// TwinCAT 3 PLC project PLC
// ProgramVersion: 3.1.4023.0
// libraries:
//   Tc2_ControllerToolbox, * (Beckhoff Automation GmbH)
//   Tc2_EtherCAT, * (Beckhoff Automation GmbH)
//   Tc2_FTP, * (Beckhoff Automation GmbH)
//   Tc2_ModbusRTU, * (Beckhoff Automation GmbH)
//   Tc2_ModbusSrv, * (Beckhoff Automation GmbH)
//   Tc2_ProfinetDiag, * (Beckhoff Automation GmbH)
//   Tc2_Standard, * (Beckhoff Automation GmbH)
//   Tc2_SUPS, * (Beckhoff Automation GmbH)
//   Tc2_System, * (Beckhoff Automation GmbH)
//   Tc2_Utilities, * (Beckhoff Automation GmbH)
//   Tc3_EventLogger, * (Beckhoff Automation GmbH)
//   Tc3_IotBase, * (Beckhoff Automation GmbH)
//   Tc3_JsonXml, * (Beckhoff Automation GmbH)
//   Tc3_Module, * (Beckhoff Automation GmbH)
//   Base Interfaces,newest,System
// project tree:
//   DUTs/Enums/ eGridTripMode.TcDUT, eBatteryType.TcDUT, eObject_ID.TcDUT, ePNcouplerType.TcDUT, eSubValues.TcDUT, Phases.TcDUT
//   DUTs/Structs/ ST_AnalogInputData.TcDUT, ST_AnalogInputDiag.TcDUT
//   DUTs/System/ ST_System_Config.TcDUT, ST_System_GridcodeParams.TcDUT, ST_System_MachineParams.TcDUT
//   GVLs/ GVL.TcGVL, Settings.TcGVL, Units.TcGVL
//   / PlcTask.TcTTO, MonitorControlTask.TcTTO
//   POUs/Datalogger/DataLogging/ ArrayVariables.TcPOU, Datalogger.TcPOU, ST_Datalog_event.TcDUT
//   POUs/Datalogger/FUNCTIONBLOCKS/ FB_CSVWriter.TcPOU, FB_Datalogger.TcPOU, ToHexConverter.TcPOU
//   POUs/ErrorHandling/ ErrorHandling.TcPOU, FB_AddErrorST.TcPOU
//   POUs/ErrorHandling/New eventlogger %28TBD%29/ EventLogger.TcPOU (not stored), FB_Alarm.TcPOU (not stored), fb_EventAlarm.TcPOU (not stored)
//   POUs/ErrorHandling/_enums/ eErrAckAccess.TcDUT, eSeverity.TcDUT
//   POUs/ErrorHandling/_strucs/ ST_ErrorStruct.TcDUT
//   POUs/EventLogger/ EventLog.TcPOU (excluded from build), WriteLogItem.TcPOU (excluded from build)
//   POUs/EventLogger/_enums/ eLogSeverity.TcDUT
//   POUs/EventLogger/_Structs/ ST_EventLoggerParams.TcDUT
//   POUs/Functions-FBs-Programs/ Fb_BindControlVars.TcPOU, FB_OverCurrentDetect.TcPOU, fb_Ramp_dual.TcPOU, fbValueOutOfRange.TcPOU, fb_IncrementPowerStep.TcPOU, fb_Ramp.TcPOU, FB_UpperLimitAndTimeExceeded.TcPOU
//   POUs/Functions-FBs-Programs/IO_modules/Beckhoff/ FB_EK1100.TcPOU, FB_EL34xx.TcPOU, FB_EL3453.TcPOU
//   POUs/Functions-FBs-Programs/IO_modules/Beckhoff/Structs/ DataSelector.TcDUT, ST_EL34xx_PhaseStatus.TcDUT, ST_EL34xx_TotalStatus.TcDUT
//   POUs/Functions-FBs-Programs/IO_modules/Wago/ FB_Wago750354_BusCoupler.TcPOU, FB_Wago750495_PowerMonitor.TcPOU
//   POUs/Functions-FBs-Programs/IO_modules/Wago/Structs/Wago750354/ ST_Wago750354_get.TcDUT
//   POUs/Functions-FBs-Programs/IO_modules/Wago/Structs/Wago750495/ eWago750495_ACDataID.TcDUT, eWago750495_HarmonicsDataID.TcDUT, eWago750495_MeasureGroupID.TcDUT, eWago750495_StatDataID.TcDUT, ST_Wago750495_Data.TcDUT, ST_Wago750495_ExtStatusWord.TcDUT, ST_Wago750495_Get.TcDUT, ST_Wago750495_Set.TcDUT, ST_Wago750495_StatusWord.TcDUT
//   POUs/Functions-FBs-Programs/_acFunctions/ AcCheck.TcPOU, ACFrequencyCheck.TcPOU, ACVoltageCheck.TcPOU, CurrentToKw.TcPOU, fb_LOMdetection.TcPOU, kWToCurrent.TcPOU, LineUnbalance.TcPOU, PowerFactor.TcPOU, ReactivePower.TcPOU
//   POUs/Functions-FBs-Programs/_generalFunctions/ Between.TcPOU, ConcatMultiString.TcPOU, fb_MovingAverage.TcPOU, FB_StartStop.TcPOU, F_RoundReal.TcPOU, IsNaN.TcPOU, LimitTrigger.TcPOU, PackByte.TcPOU, PackWord.TcPOU, Median.TcPOU, Scale.TcPOU, ValueOutOfRange.TcPOU, WriteOnEdge.TcPOU, XNOR.TcPOU
//   POUs/Functions-FBs-Programs/_PRGS/ SystemClock.TcPOU
//   POUs/ MAIN_Fast.TcPOU, MAIN_Slow.TcPOU
//   POUs/MonitoringControl/ ControlManager.TcPOU, FB_TestScripts.TcPOU
//   POUs/MonitoringControl/HMI/ FB_HMIButtons.TcPOU, HMI.TcPOU
//   POUs/MonitoringControl/HMI/_Structs/ControlStructures/HardSettings %28localOnly%29/ ST_HardSettings.TcDUT (not stored), ST_HardSettings_DCcharger.TcDUT (not stored), ST_HardSettings_ParallelOperation.TcDUT (not stored), ST_HardSettings_PeakshaveBox.TcDUT (not stored), ST_HardSettings_Setup.TcDUT (not stored), ST_HardSettings_System.TcDUT (not stored)
//   POUs/MonitoringControl/HMI/_Structs/ControlStructures/OperationVars/ ST_OperationVars.TcDUT, ST_OperationVars_BMS.TcDUT, ST_OperationVars_DCcharger.TcDUT, ST_OperationVars_Genset.TcDUT, ST_OperationVars_Grid.TcDUT, ST_OperationVars_ParallelOperation.TcDUT, ST_OperationVars_System.TcDUT
//   POUs/MonitoringControl/HMI/_Structs/ControlStructures/SoftSettings %28Local+Extern%29/NestedStructs/ ST_Genset_params.TcDUT (not stored), ST_Genset_setpoints.TcDUT (not stored), ST_Input_breakersettings.TcDUT (not stored), ST_Loadbank_params.TcDUT (not stored), ST_peakshave_setpoints.TcDUT (not stored), ST_ScheduleTimeSlot.TcDUT (not stored)
//   POUs/MonitoringControl/HMI/_Structs/ControlStructures/SoftSettings %28Local+Extern%29/ ST_SoftSettings.TcDUT (not stored), ST_Softsettings_AcDcCharger.TcDUT (not stored), ST_SoftSettings_Genset.TcDUT (not stored), ST_SoftSettings_Grid.TcDUT (not stored), ST_SoftSettings_PeakshaveBox.TcDUT (not stored), ST_SoftSettings_Setup.TcDUT (not stored), ST_SoftSettings_System.TcDUT (not stored)
//   POUs/MonitoringControl/HMI/_Structs/ControlStructures/ ST_ControlsHMIonly.TcDUT, ST_ControlVars.TcDUT
//   POUs/MonitoringControl/HMI/_Structs/MonitoringStructures/ ST_HMIdata.TcDUT, ST_HMI_ConditionalFormatting.TcDUT, ST_HMI_Monitor_AcDcCharger.TcDUT, ST_HMI_Monitor_Arraydata.TcDUT, ST_HMI_Monitor_ArrayDataFormat.TcDUT, ST_HMI_Monitor_Connections.TcDUT, ST_HMI_Monitor_Battery.TcDUT, ST_HMI_Monitor_CoolingSystem.TcDUT, ST_HMI_Monitor_Enclosure.TcDUT, ST_HMI_Monitor_FireDetection.TcDUT, ST_HMI_Monitor_IPSU.TcDUT, ST_HMI_Monitor_Limits.TcDUT, ST_HMI_Monitor_OCP.TcDUT, ST_HMI_Monitor_Powerstack.TcDUT, ST_HMI_Monitor_Protections.TcDUT, ST_HMI_Monitor_PSB.TcDUT, ST_HMI_Monitor_switchgear.TcDUT, ST_HMI_Monitor_System.TcDUT, ST_HMI_Monitor_UPS.TcDUT, ST_HMI_Monitor_ZPT.TcDUT, ST_HMI_PowerMeas.TcDUT, ST_HMI_PowerMeasDC.TcDUT
//   POUs/MonitoringControl/HMI/_Structs/ ST_HMI_Control.TcDUT, ST_HMI_Historize.TcDUT, ST_HMI_Monitor.TcDUT
//   POUs/MonitoringControl/IoT/DUTS/ eConnectionState.TcDUT, eDataMappingVarNames.TcDUT, eIoTCommVersion.TcDUT, eLogType.TcDUT, eUpdate.TcDUT, e_ORAttributeType.TcDUT, ST_AutoProvisioning.TcDUT, ST_IotProps.TcDUT, ST_RW.TcDUT, ST_Supervisor.TcDUT, ST_VarBuffer.TcDUT
//   POUs/MonitoringControl/IoT/ FB_IotController.TcPOU, MqttComOpenremote.TcPOU, RestComOpenremote.TcPOU
//   POUs/MonitoringControl/IoT/_Structs/ ST_IoTDataHMI.TcDUT, ST_IotData_credits.TcDUT, st_IOT_params.TcDUT, ST_IOT_SentStateLog.TcDUT
//   POUs/MonitoringControl/ProfinetController/enums/ eExternalControlMode.TcDUT, GenGridMode.TcDUT, uSWversion.TcDUT
//   POUs/MonitoringControl/ProfinetController/ FB_ExtControllerTest.TcPOU, FB_ExternalController.TcPOU
//   POUs/MonitoringControl/ProfinetController/Structs/future use/ ST_PNInput_DCBusExpansion.TcDUT, ST_PNInput_DCCharger.TcDUT, ST_PNInput_ParallelOperation.TcDUT, ST_PNOutput_DCCharger.TcDUT, ST_PNOutput_DCExpansion.TcDUT, ST_PNOutput_ParallelOperation.TcDUT
//   POUs/MonitoringControl/ProfinetController/Structs/NestedStructs/ ST_PNInput_ACDCCharger.TcDUT, ST_PNInput_Battery.TcDUT, ST_PNInput_GenControl.TcDUT, ST_PNInput_General.TcDUT, ST_PNInput_InputField.TcDUT, ST_PNInput_InputGridControl.TcDUT, ST_PNInput_PeakShaveBox.TcDUT, ST_PNInput_Powerstack.TcDUT, ST_PNOutput_ACDCCharger.TcDUT, ST_PNOutput_Battery.TcDUT, ST_PNOutput_GenControl.TcDUT, ST_PNOutput_General.TcDUT, ST_PNOutput_InputField.TcDUT, ST_PNOutput_InputGridControl.TcDUT, ST_PNOutput_OutputField.TcDUT, ST_PNOutput_PeakShaveBox.TcDUT, ST_PNOutput_PowerStack.TcDUT, ST_PNOutput_ZPT.TcDUT
//   POUs/MonitoringControl/ProfinetController/Structs/ ST_PNcontroller_params.TcDUT, ST_PNinput.TcDUT, ST_PNOutput.TcDUT, ST_PNTest.TcDUT
//   POUs/MonitoringControl/_Enums/ eAcInputType.TcDUT, eCapTestSTate.TcDUT, eControlSources.TcDUT, eDcInputType.TcDUT, eEarthingSystems.TcDUT, eGridFormingMode.TcDUT, eGridMode.TcDUT, eNetContactorDirection.TcDUT, eOperationMode.TcDUT, ePeakshaveMode.TcDUT, eSchedulerMode.TcDUT, ePowerControlType.TcDUT, eSystemState.TcDUT, eUgridPowerMode.TcDUT
//   POUs/MonitoringControl/_Structs/ ST_ExtController_Events.TcDUT, ST_ExtController_get.TcDUT, ST_ExtController_limits.TcDUT, ST_ExtController_Set.TcDUT, ST_PLCPersistentVars.TcDUT
//   POUs/Objects/4Grouter/ FB_Teltonika.TcPOU
//   POUs/Objects/4Grouter/Struct/ dwtoreal.TcDUT, eModemState.TcDUT, eNetworkState.TcDUT, eSimSelectionMode.TcDUT, eSimState.TcDUT, eSMSStatus.TcDUT, eWifiSecurityTypes.TcDUT, eWifiStatus.TcDUT, st_Device.TcDUT, st_GPS.TcDUT, st_mobile.TcDUT, st_router_get.TcDUT, ST_Router_params.TcDUT, st_Router_Events.TcDUT, ST_Router_set.TcDUT, st_Wifi.TcDUT
//   POUs/Objects/ACDCCharger/Enums/ eAcDcChargerState.TcDUT
//   POUs/Objects/ACDCCharger/ FB_ACDCcharger.TcPOU
//   POUs/Objects/ACDCCharger/Structs/Hadi/ E_ChargerState.TcDUT, ST_CanId.TcDUT, ST_ChargerControl.TcDUT, ST_Control.TcDUT, ST_Data.TcDUT, ST_ModuleControl.TcDUT, ST_ModuleData.TcDUT, ST_ModuleStatus.TcDUT
//   POUs/Objects/ACDCCharger/Structs/ ST_ACDCCharger_events.TcDUT, ST_ACDCCharger_get.TcDUT, ST_ACDCCharger_params.TcDUT, ST_ACDCCharger_set.TcDUT, ST_SystemDiagnostic.TcDUT, ST_SystemEval.TcDUT
//   POUs/Objects/ACSwitchgear %28clientbox%29/ FB_ACSwitchgear.TcPOU (not stored), ST_ACswitchgear_events.TcDUT (not stored), ST_ACSwitchgear_Get.TcDUT (not stored), ST_ACswitchgear_IO.TcDUT (not stored), ST_ACswitchgear_params.TcDUT (not stored), ST_ACswitchgear_set.TcDUT (not stored)
//   POUs/Objects/BMS/eNums/ eBMS_Status.TcDUT, eHVDC_Powerstatus.TcDUT, ePOUState.TcDUT, ePowerControl.TcDUT, ePowerOnStatus.TcDUT
//   POUs/Objects/BMS/ FB_BMS.TcPOU, FB_BMS_IO.TcPOU
//   POUs/Objects/BMS/Structs/ st_BMS_Events.TcDUT, st_BMS_Get.TcDUT, st_BMS_Params.TcDUT, st_BMS_BatterySummary.TcDUT, st_BMS_Set.TcDUT, st_MBMU_BatterySummary.TcDUT, st_MBMU_Status.TcDUT, st_SBMU_BatterySummary.TcDUT, st_SBMU_Status.TcDUT
//   POUs/Objects/CoolingSystem/ FB_CoolingSystem.TcPOU, FB_CoolingSystem_IO.TcPOU
//   POUs/Objects/CoolingSystem/HeatpumpSystem/eNums/ eHeatPumpMode.TcDUT, eHeatPumpState.TcDUT, eSupportedHeatpumps.TcDUT
//   POUs/Objects/CoolingSystem/HeatpumpSystem/ FB_HeatPumpSystem.TcPOU, FB_LGHeatpump.TcPOU, FB_TraneHeatpump.TcPOU, IF_Heatpump.TcIO
//   POUs/Objects/CoolingSystem/HeatpumpSystem/Structs/ LG_Coils.TcDUT, LG_ControlRegs.TcDUT, LG_get.TcDUT, LG_InputRegs.TcDUT, LG_set.TcDUT, LG_Statusbits.TcDUT, ST_HeatpumpData.TcDUT, ST_HeatPumpEvents.TcDUT, ST_HeatPump_Get.TcDUT, ST_HeatPumpSystemEvents.TcDUT, ST_HeatpumpSystemGet.TcDUT, st_OperatingPoint.TcDUT
//   POUs/Objects/CoolingSystem/_Enum/ eConditioningRequirement.TcDUT, eCoolingSystemState.TcDUT, ePumpState.TcDUT, eCoolingControl.TcDUT, eCoolingPowerRequest.TcDUT
//   POUs/Objects/CoolingSystem/_Structs/ ST_ConditioningRequirements.TcDUT, ST_CoolingSystem_Control.TcDUT, ST_CoolingSystem_Events.TcDUT, ST_CoolingSystem_Get.TcDUT, ST_CoolingSystem_Inputs.TcDUT, ST_CoolingSystem_Outputs.TcDUT, ST_Coolingsystem_params.TcDUT
//   POUs/Objects/DCSwitchgear/ FB_DCSwitchgear.TcPOU, ST_DCSwitchgear_Get.TcDUT
//   POUs/Objects/Enclosure/Climate/ FB_EnclosureClimate.TcPOU, ST_Enclosureclimate_events.TcDUT, ST_EnclosureClimate_get.TcDUT, ST_EnclosureClimate_Params.TcDUT
//   POUs/Objects/Enclosure/Doors/ FB_DoorsNLocks.TcPOU, ST_DoorsNLocks_get.TcDUT
//   POUs/Objects/Enclosure/ FB_Enclosure.TcPOU
//   POUs/Objects/Enclosure/LedIndicator/ArduinoController/ FB_LedArduino.TcPOU
//   POUs/Objects/Enclosure/LedIndicator/BeckhoffController/ eDCstate.TcDUT, eLEDSteps.TcDUT, FB_LedBeckhoff.TcPOU, LEDColor.TcDUT, LEDCommands.TcDUT, LEDControl.TcDUT, LEDStatus.TcDUT, eSystemStatus.TcDUT
//   POUs/Objects/Enclosure/LedIndicator/ eColorOrder.TcDUT, FB_Ledstrip.TcPOU, ST_Ledstrip_get.TcDUT, st_Ledstrip_MachineData.TcDUT, st_Ledstrip_params.TcDUT
//   POUs/Objects/Enclosure/_struct/ ST_Enclosure_get.TcDUT, st_Enclosure_params.TcDUT, ST_enclosure_set.TcDUT
//   POUs/Objects/GenComm/eNums/ eGenControlProtocol.TcDUT, eGenOperationMode.TcDUT, eOnOffState.TcDUT
//   POUs/Objects/GenComm/ FB_AGC150.TcPOU, FB_GenComm.TcPOU
//   POUs/Objects/GenComm/Structs/ ST_Genset_Get.TcDUT, ST_AGC150_Set.TcDUT, ST_GenComm_Params.TcDUT, ST_Genset_Set.TcDUT
//   POUs/Objects/HartingIO/ FB_HartingIO.TcPOU, ST_HartingIO_get.TcDUT, ST_HartingIO_params.TcDUT, ST_HartingIO_set.TcDUT
//   POUs/Objects/HartingIO/_Enum/ eAOTarget.TcDUT, eOutputContactSignal.TcDUT, eInputSignal.TcDUT
//   POUs/Objects/InterMachineCom/ FB_ConnectMqttBroker.TcPOU, FB_InterMachineCommunication.TcPOU, ST_InterMachineCom_Master.TcDUT, ST_IntermachineCom_params.TcDUT, st_InterMachineCom_Slave.TcDUT, ST_InterMachineCom_SlaveConData.TcDUT
//   POUs/Objects/InternalPowerSupply/eNums/ e400VSupplySource.TcDUT, eSupplyState.TcDUT
//   POUs/Objects/InternalPowerSupply/ FB_InternalPowerSupply.TcPOU, FB_InternalPowerSupply_IO.TcPOU
//   POUs/Objects/InternalPowerSupply/Structs/ ST_InternalPowerStatus.TcDUT, ST_InternalPowerSupply_Events.TcDUT, ST_InternalPowerSupply_Get.TcDUT, ST_InternalPowerSupply_Params.TcDUT, ST_InternalPowerSupply_PowerDemand.TcDUT
//   POUs/Objects/InternalPowerSupply/UPS/eNums/ eUPSState.TcDUT
//   POUs/Objects/InternalPowerSupply/UPS/ FB_UPS.TcPOU
//   POUs/Objects/InternalPowerSupply/UPS/Structs/ ST_UPSData.TcDUT, ST_UPSEvents.TcDUT, ST_UPSGET.TcDUT
//   POUs/Objects/NeutralTransformer/ FB_NeutralTransformer.TcPOU, FB_NeutralTransformer_IO.TcPOU
//   POUs/Objects/NeutralTransformer/InternalPowerSupply/eNums/ e400VSupplySource.TcDUT (not stored), eSupplyState.TcDUT (not stored)
//   POUs/Objects/NeutralTransformer/InternalPowerSupply/ FB_InternalPowerSupply.TcPOU (not stored), FB_InternalPowerSupply_IO.TcPOU (not stored)
//   POUs/Objects/NeutralTransformer/InternalPowerSupply/Structs/ ST_InternalPowerStatus.TcDUT (not stored), ST_InternalPowerSupply_Events.TcDUT (not stored), ST_InternalPowerSupply_Get.TcDUT (not stored), ST_InternalPowerSupply_Params.TcDUT (not stored), ST_InternalPowerSupply_PowerDemand.TcDUT (not stored), ST_InternalPowersupply_set.TcDUT (not stored)
//   POUs/Objects/NeutralTransformer/InternalPowerSupply/UPS/eNums/ eUPSState.TcDUT (not stored)
//   POUs/Objects/NeutralTransformer/InternalPowerSupply/UPS/ FB_UPS.TcPOU (not stored)
//   POUs/Objects/NeutralTransformer/InternalPowerSupply/UPS/Structs/ ST_UPSData.TcDUT (not stored), ST_UPSEvents.TcDUT (not stored), ST_UPSGET.TcDUT (not stored)
//   POUs/Objects/NeutralTransformer/_Struct/ ST_NeutralTransformer_events.TcDUT, ST_NeutralTransformer_Get.TcDUT, ST_Neutraltransformer_params.TcDUT
//   POUs/Objects/PeakshaveBox/DUTs/ ePsbCtRange.TcDUT (excluded from build), ePSBMode.TcDUT, ePSBhardware.TcDUT, ST_PowerMeasurement_status.TcDUT, eWago750495_ACDataID_1.TcDUT, eWago750495_HarmonicsDataID_1.TcDUT, eWago750495_MeasureGroupID_1.TcDUT, eWago750495_StatDataID_1.TcDUT, ST_Wago750495_Data_1.TcDUT, ST_Wago750495_ExtStatusWord_1.TcDUT, ST_Wago750495_Read_1.TcDUT, ST_Wago750495_StatusWord_1.TcDUT, ST_Wago750495_Write_1.TcDUT
//   POUs/Objects/PeakshaveBox/ ST_peakshavebox_params.TcDUT, ST_PeakshaveBox_Set.TcDUT, FB_PeakshaveBox.TcPOU, ST_PeakShaveBox_Get.TcDUT
//   POUs/Objects/PLCStatus/Enum/ eFTPState.TcDUT, eNetcomState.TcDUT, eInstalState.TcDUT
//   POUs/Objects/PLCStatus/ FB_PLCState.TcPOU, FB_PLCUpdate.TcPOU, ST_EL9410.TcDUT, ST_PLCstate_get.TcDUT, ST_PLC_events.TcDUT
//   POUs/Objects/PowerQualityMonitor/FB_Janitza_UMG801/ FB_Janitza.TcPOU, PowerMeterConfig.TcGVL
//   POUs/Objects/PowerQualityMonitor/ FB_PowerQualityMonitoring.TcPOU
//   POUs/Objects/PowerQualityMonitor/_Enums/ eACRotationState.TcDUT
//   POUs/Objects/PowerQualityMonitor/_Structs/ ST_MeasurementFieldData.TcDUT, ST_MeasurementVoltageData.TcDUT, ST_PowerMonitor_BESS.TcDUT, ST_PowerMonitor_Events.TcDUT, ST_PowerMonitor_get.TcDUT, ST_PowerMonitor_InputField.TcDUT, ST_PowerMonitor_OutputField.TcDUT
//   POUs/Objects/PowerStack/NetContactor/ eNetcontMode.TcDUT, FB_NetContactor.TcPOU, FB_NetContactor_IO.TcPOU
//   POUs/Objects/PowerStack/NetContactor/_Structs/ ST_Netcontactor_Events.TcDUT, ST_Netcontactor_get.TcDUT, ST_Netcontactor_set.TcDUT
//   POUs/Objects/PowerStack/PowerModule/ FB_Powermodule_additionalMeasurements.TcPOU, FB_PowerModule.TcPOU, FB_PowerModule_Buscoupler.TcPOU, FB_PowerModule_Inverter.TcPOU
//   POUs/Objects/PowerStack/_Enums/ eInverterModes.TcDUT, eNetContactorState.TcDUT, ePowerModes.TcDUT, ePowerModuleThrottlingState.TcDUT, ePowerstate.TcDUT, eStatusPowerModule.TcDUT, eStatusPowerStack.TcDUT, ePLM.TcDUT
//   POUs/Objects/PowerStack/ FB_PowerStack.TcPOU
//   POUs/Objects/PowerStack/_Structs/NestedStructs/ ST_Powermodule_CalibData.TcDUT, ST_InverterControlWord.TcDUT, ST_Inverter_StatusWord.TcDUT, ST_Inverter_UgridStatusWord.TcDUT, ST_Inverter_additionalTemperatures.TcDUT, ST_Inverter_LineState.TcDUT, ST_Inverter_Write.TcDUT, ST_Powermodule_Events.TcDUT, ST_Powermodule_PowerCurveCoefficients.TcDUT, ST_PowerStack_Events.TcDUT, ST_Powerstack_ShiftingParams.TcDUT
//   POUs/Objects/PowerStack/_Structs/ ST_PowerModule_calibration.TcDUT, ST_PowerModule_params.TcDUT, ST_PowerModule_get.TcDUT, ST_PowerModule_set.TcDUT, ST_Powerstack_Calibration.TcDUT, ST_PowerStack_get.TcDUT, ST_Powerstack_LOMParams.TcDUT, ST_PowerStack_params.TcDUT, ST_PowerStack_Set.TcDUT
//   POUs/Objects/ProtectionSystems/ FB_ProtectionSystems.TcPOU
//   POUs/Objects/ProtectionSystems/FireDetection/ FB_FireDetection.TcPOU, FB_FireDetection_IO.TcPOU
//   POUs/Objects/ProtectionSystems/FireDetection/_Enums/ eCOAlarmStatus.TcDUT, eSmokeDetectAlarmStatus.TcDUT
//   POUs/Objects/ProtectionSystems/FireDetection/_Structs/ ST_CODetectors.TcDUT, ST_FireDetection_get.TcDUT, st_Firedetection_params.TcDUT, ST_FireDetection_set.TcDUT, ST_FireSystem_Events.TcDUT, ST_SmokeDetectors.TcDUT, ST_SmokeDetIO.TcDUT
//   POUs/Objects/ProtectionSystems/InsulationMonitoring/ FB_InsulationMonitor.TcPOU
//   POUs/Objects/ProtectionSystems/InsulationMonitoring/_Structs/ ST_InsulationMonitor_get.TcDUT, ST_InsulationMonitor_params.TcDUT, St_InsulationMonitor_PassThrough.TcDUT, ST_InsulationMonitor_set.TcDUT
//   POUs/Objects/ProtectionSystems/OvercurrentProtection/ FB_OvercurrentProtection.TcPOU
//   POUs/Objects/ProtectionSystems/OvercurrentProtection/_Structs/ ST_OvercurrentProtection_Events.TcDUT, ST_OvercurrentProtection_get.TcDUT, ST_OvercurrentProtection_InternalLinking.TcDUT, ST_OvercurrentProtection_Params.TcDUT, ST_OvercurrentProtection_set.TcDUT
//   POUs/Objects/ProtectionSystems/ResidualCurrentMonitoring/ FB_RCMonitor.TcPOU
//   POUs/Objects/ProtectionSystems/ResidualCurrentMonitoring/_Structs/ ST_ResidualCurrentMonitor_get.TcDUT
//   POUs/Objects/ProtectionSystems/SurgeProtection/ FB_SurgeProtection.TcPOU
//   POUs/Objects/ProtectionSystems/SurgeProtection/_Structs/ ST_Surgeprotection_get.TcDUT
//   POUs/Objects/ProtectionSystems/_Struct/ ST_ProtectionSystems_get.TcDUT, ST_ProtectionSystems_Params.TcDUT, ST_ProtectionSystems_set.TcDUT
//   POUs/Objects/WearLogging/ eEntryType.TcDUT, eLogItemGroupID.TcDUT, eLogTypes.TcDUT, FB_Varlogger.TcPOU, LogState.TcDUT, WearLogging.TcPOU
//   POUs/Safety/ Safety.TcPOU, ST_Safety_ContactorEDM.TcDUT, ST_Safety_get.TcDUT, ST_Safety_ToSafetyPrg.TcDUT
//   POUs/System/ FB_SystemControl.TcPOU
//   POUs/System/GenGridControl/ FB_ContactorControl.TcPOU, FB_GenGridController.TcPOU
//   POUs/System/GenGridControl/_enums/ eBreakerOperationMode.TcDUT, eGenIsoInverterMode.TcDUT, eGensetStartStop.TcDUT, eGensetMode.TcDUT, ePowerControlMode.TcDUT, eGenGridState.TcDUT, eRunCondition.TcDUT
//   POUs/System/GenGridControl/_structs/ ST_ContactorControl_params.TcDUT, ST_GenGridController_Events.TcDUT, ST_GenGridController_get.TcDUT, ST_GenGridController_Params.TcDUT, St_GenGridController_ParamsGenset.TcDUT, ST_GenGridController_SyncData.TcDUT
//   POUs/System/PowerControl/ FB_PowerControl.TcPOU, fb_measurementCheck.TcPOU
//   POUs/System/PowerControl/_enums/ ePIDmode.TcDUT
//   POUs/System/PowerControl/_Structs/ ST_PowerControl_Events.TcDUT, ST_PowerControl_Get.TcDUT, st_Powercontrol_params.TcDUT, st_Powercontrol_PIDparams.TcDUT, ST_PowerControl_PsTarget_Measurements.TcDUT, ST_Powercontrol_set.TcDUT, ST_PowerControl_SocDroopParams.TcDUT, ST_PowerControl_Target.TcDUT
//   POUs/System/_Structs/ ST_SystemTime.TcDUT, ST_System_Calibration.TcDUT, ST_System_Events.TcDUT, ST_System_params.TcDUT, ST_System_Properties.TcDUT, ST_System_set.TcDUT, ST_System_get.TcDUT, ST_System_Monitor.TcDUT, ST_System_Control.TcDUT

CONFIGURATION PLC
    RESOURCE PLC ON TwinCAT3
        TASK PlcTask(INTERVAL := T#2ms, PRIORITY := 4);
        TASK MonitorControlTask(INTERVAL := T#10ms, PRIORITY := 8);
        PROGRAM MAIN_Fast WITH PlcTask : MAIN_Fast;
        PROGRAM MAIN_Slow WITH MonitorControlTask : MAIN_Slow;
    END_RESOURCE
END_CONFIGURATION

// ---- DUTs/Enums/eGridTripMode.TcDUT
{attribute 'qualified_only'}
{attribute 'strict'}
TYPE eGridTripMode :
(
	Gridcode := 500,
	Default	:= 30,
	UPS		:= 10	
) UINT; //milliseconds
END_TYPE

// ---- DUTs/Enums/eBatteryType.TcDUT
{attribute 'qualified_only'}
{attribute 'strict'}
TYPE eBatteryType :
(
	standard_306Ah := 0,
	highpower_280Ah := 1
);
END_TYPE

// ---- DUTs/Enums/eObject_ID.TcDUT
{attribute 'qualified_only'}
{attribute 'to_string'}
TYPE eObject_ID :
(	
	None					:= 0,
	Safety					:= 10,
	PowerStack				:= 100,
	NetContactor			:= 150,
	PowerModuleMaster 		:= 200,
	PowerModuleSlave 		:= 300,
	PowerMonitor			:= 400,
	InternalPowerSupply		:= 500,
	UPS						:= 550,
	NeutralTransformer		:= 600,
	HartingIO				:= 650,
	Battery					:= 700,
	Cooling					:= 800,
	HeatPump				:= 850,
	AC_Switchgear			:= 900,
	DC_Switchgear			:= 950,
	RCM						:= 1000,
	SurgeProtection			:= 1010,
	InsulationMonitor		:= 1020,
	Firedetection			:= 1030,
	OCP						:= 1050,
	Enclosure_LED			:= 1200,
	Enclosure_doors			:= 1210,
	Enclosure_climate		:= 1220,
	PLC						:= 2000,
	Router					:= 2100,
	PNcontroller			:= 2200,
	IotController			:= 2300,
	PeakshaveBox			:= 2400,
	ACDCCharger				:= 2500,
	GenGridController		:= 3000,
	PowerController			:= 3100,
	System					:= 3200,
	Genset					:= 4000
	
) WORD := None;
END_TYPE

// ---- DUTs/Enums/ePNcouplerType.TcDUT
{attribute 'qualified_only'}
{attribute 'strict'}

TYPE ePNcouplerType :
(
	None := 0,
	ModbusTCP:= 1,
	Profinet := 2,
	ModbusTCPV2 := 3
);
END_TYPE

// ---- DUTs/Enums/eSubValues.TcDUT
{attribute 'qualified_only'}
{attribute 'strict'}
TYPE eSubValues :
(
	Minimum := 0,
	Average := 1,
	Maximum := 2
);
END_TYPE

// ---- DUTs/Enums/Phases.TcDUT
{attribute 'qualified_only'}
{attribute 'strict'}
{attribute 'to_string'}
TYPE Phases :
(
	AVG 		:= 0,
	L1 			:= 1,
	L2 			:= 2,
	L3 			:= 3,
	N 			:= 4,
	minimum		:= 5,
	maximum		:= 6
) INT;
END_TYPE

// ---- DUTs/Structs/ST_AnalogInputData.TcDUT
TYPE ST_AnalogInputData :
STRUCT
	Value			: INT;
	Status			: ST_AnalogInputDiag;
END_STRUCT
END_TYPE

// ---- DUTs/Structs/ST_AnalogInputDiag.TcDUT
TYPE ST_AnalogInputDiag :
STRUCT
	Underrange			: BIT;
	Overrange			: BIT;
	Error				: BIT;
END_STRUCT 
END_TYPE

// ---- DUTs/System/ST_System_Config.TcDUT
TYPE ST_System_Config :
STRUCT
	DefaultSettingsActive			: BOOL := TRUE; //To verify when all settings have been reset.
	b_DoublePowerModule				: BOOL := FALSE;
	b_PeakshaverBoxEnable			: BOOL := FALSE;
	
	//NeutralTransformer
	b_NeutralTransformer			: BOOL := FALSE;
	
	
	//Netcontactor
	b_AutomaticACrotation			: BOOL := FALSE;
	
	//DC
	b_DCbuscoupling					: BOOL := FALSE;
	b_DcCharger						: BOOL := FALSE;
	
	//AC
	b_ACInputConnection				: BOOL := FALSE;
	b_ThirdOutputConnection			: BOOL := FALSE;
	//communication
	e_PNcouplerType					: ePNcouplerType := ePNcouplerType.None;
	
	//batteries
	by_NoBatteryStrings			 	: BYTE := 3; // pieces
	e_BatteryType					: eBatteryType := eBatteryType.standard_306Ah;
	
	//Powernet option
	b_PowernetClient				: BOOL :=  FALSE;
	
	//CLIENT specifics
	b_ClientHMI						: BOOL := FALSE;
	
END_STRUCT
END_TYPE

// ---- DUTs/System/ST_System_GridcodeParams.TcDUT
TYPE ST_System_GridcodeParams :
STRUCT
	r_GridNominalVoltage				: REAL := 400; //VAC
	r_GridNominalFrequency				: REAL := 50; // Hz
	r_GridVoltageMin					: REAL := 360;
	r_GridvoltageMax					: REAL := 440;
	r_GridFrequencyMin					: REAL := 48.5;
	r_GridFrequencyMax					: REAL := 51.5;
	r_CurrentUnbalanceLimit				: REAL := 50;  //%
	ui_GCokReleaseTime					: UINT := 60; //seconds
	ui_GCTripMaxTripTime				: UINT := 40; // milliseconds
END_STRUCT
END_TYPE

// ---- DUTs/System/ST_System_MachineParams.TcDUT
TYPE ST_System_MachineParams :
STRUCT
	BMS									: ST_BMS_params;
	ACDCCharger							: ST_ACDCCharger_params;
	Interpowersupply					: ST_InternalPowerSupply_Params;
	Powerstack							: ST_Powerstack_Params;
	Coolingsystem						: ST_Coolingsystem_Params;
	NeutralTransformer					: ST_Neutraltransformer_Params;
	Protections							: ST_Protectionsystems_Params;
	Enclosure							: ST_Enclosure_Params;
	system								: ST_System_params;
	PNController						: ST_PNcontroller_params;
	IOT									: ST_IOT_params;
	Router								: ST_Router_params;
	PSB									: ST_peakshavebox_params;
	ACswitchgear						: ST_ACswitchgear_params;
	HartingIO							: ST_HartingIO_params;
	GenComm								: ST_GenComm_params;
	Eventlogger							: ST_EventLoggerParams;
END_STRUCT
END_TYPE

// ---- POUs/Datalogger/DataLogging/ST_Datalog_event.TcDUT
TYPE ST_Datalog_event :
STRUCT
	s_header		: STRING;
	s_data			: STRING;			
END_STRUCT
END_TYPE

// ---- POUs/ErrorHandling/_enums/eErrAckAccess.TcDUT
{attribute 'qualified_only'}
{attribute 'strict'}
TYPE eErrAckAccess :
(
	General := 0,
	Operator := 1,
	VDL := 2
);
END_TYPE

// ---- POUs/ErrorHandling/_enums/eSeverity.TcDUT
{attribute 'qualified_only'}
{attribute 'to_string'}
TYPE eSeverity :
(
	None						:= 0,
	Info						:= 1,
	Warning 					:= 2,
	NormalShutdown				:= 3,
	QuickShutdown				:= 4,
	EmergencyShutdown			:= 5 //ONLY CALL FROM SAFETY PROGRAM		
);
END_TYPE

// ---- POUs/ErrorHandling/_strucs/ST_ErrorStruct.TcDUT
TYPE ST_ErrorStruct :
STRUCT
	b_ErrorActive	:BOOL;
	s_Severity 		:STRING(20);
	w_ID			:WORD;
	s_Message		:STRING(100);
	s_DateError		:STRING(20);
	s_TimeError		:STRING(20);
	s_TimeCleared	:STRING(20);
	b_SMSEnable		:BOOL;
END_STRUCT
END_TYPE

// ---- POUs/EventLogger/_enums/eLogSeverity.TcDUT
{attribute 'qualified_only'}
{attribute 'toString'}
TYPE eLogSeverity: //EXTENDS eSeverity:
(
	Error := 6,
	Critical := 7
);
END_TYPE

// ---- POUs/EventLogger/_Structs/ST_EventLoggerParams.TcDUT
TYPE ST_EventLoggerParams :
STRUCT
	MaxFileSize			: 	UDINT 	:= 5000000; // bytes, rotation trigger threshold (~5 MB)
	MaxFileCount		: 	UINT 	:= 5; // active + archives

	LogFileName			: 	STRING	:=	'C:\Users\Administrator\Documents\ePU10Log.txt';
	LogWriteInterval	: 	TIME 	:= T#1M; // periodic flush interval
	MaxFillGrade		: 	REAL 	:= 0.9; // flush when buffer reaches this count of RamBufferSize
	EMstopWriteDelay	:	TIME	:=	T#1S;
END_STRUCT
END_TYPE

// ---- POUs/Functions-FBs-Programs/IO_modules/Beckhoff/Structs/DataSelector.TcDUT
{attribute 'qualified_only'}
{attribute 'strict'}
TYPE DataSelector :
(
	_C 		:= 0,
	_V 		:= 1,
	_P		:= 2,
	_Q		:= 3,
	_S		:= 4,
	_E		:= 5,
	_F		:= 6	
);
END_TYPE

// ---- POUs/Functions-FBs-Programs/IO_modules/Beckhoff/Structs/ST_EL34xx_PhaseStatus.TcDUT
TYPE ST_EL34xx_PhaseStatus :
STRUCT
	bit_voltageSign				: BIT;
	bit_Overvoltage				: BIT;
	bit_Overcurrent           	: BIT;
	bit_InaccurateVoltage     	: BIT;
	bit_InaccurateCurrent     	: BIT;
	bit_VoltageGuardWarning   	: BIT;
	bit_VoltageGuardError     	: BIT;
	bit_CurrentGuardWarning   	: BIT;
	bit_CurrentGuardError     	: BIT;
	bit_TxPDOToggle           	: BIT;
END_STRUCT
END_TYPE

// ---- POUs/Functions-FBs-Programs/IO_modules/Beckhoff/Structs/ST_EL34xx_TotalStatus.TcDUT
TYPE ST_EL34xx_TotalStatus :
STRUCT
	bit_SystemState						: BIT;
	bit_GridDirection					: BIT;
	bit_FrequencyGuardWarning			: BIT;
	bit_FrequencyGuardError             : BIT;
	bit_NeutralCurrentGuardWarning      : BIT;
	bit_NeutralCurrentGuardError        : BIT;
	bit_ActivePowerGuardWarning         : BIT;
	bit_ActivePowerGuardError           : BIT;
	bit_ApparentPowerGuardWarning       : BIT;
	bit_ApparentPowerGuardError         : BIT;
	bit_PowerQualityGuardWarning        : BIT;
	bit_PowerQualityGuardError          : BIT;
	bit_TxPDOState                      : BIT;
	bit_TxPDOToggle                     : BIT;
	r_PowerQualityFactor				: REAL;
END_STRUCT
END_TYPE

// ---- POUs/Functions-FBs-Programs/IO_modules/Wago/Structs/Wago750354/ST_Wago750354_get.TcDUT
TYPE ST_Wago750354_get :
STRUCT
	b_SlaveReady							: BOOL;
END_STRUCT
END_TYPE

// ---- POUs/Functions-FBs-Programs/IO_modules/Wago/Structs/Wago750495/eWago750495_ACDataID.TcDUT
{attribute 'qualified_only'}
{attribute 'strict'}
{attribute 'to_String'}
TYPE eWago750495_ACDataID :
(
	//only RMS and peak values are declared
	//Voltages
	VoltageL1N_RMS			:= 4,
	VoltageL2N_RMS 			:= 5,
	VoltageL3N_RMS			:= 6,
	VoltageL1L2_RMS			:= 31,
	VoltageL2L3_RMS 		:= 32,
	VoltageL3L1_RMS			:= 33,
	VoltageL1N_Peak 		:= 91,
	VoltageL2N_Peak 		:= 92,
	VoltageL3N_Peak 		:= 93,
	
	//Currents
	CurrentL1_RMS			:= 1,
	CurrentL2_RMS			:= 2,
	CurrentL3_RMS			:= 3,
	CurrentN_RMS			:= 97,
	CurrentL1_Peak			:= 94,
	CurrentL2_Peak			:= 95,
	CurrentL3_Peak			:= 96,
	                           
	//Power                    
	ActivePowerL1			:= 07,
	ActivePowerL2			:= 08,
	ActivePowerL3			:= 09,
	ReactivePowerL1			:= 10,
	ReactivePowerL2			:= 11,
	ReactivePowerL3			:= 12,
	ApparentPowerL1			:= 13,
	ApparentPowerL2			:= 14,
	ApparentPowerL3			:= 15,
	
	//Energy
	ActiveEnergyTotal			:= 73,
	ActiveEnergyImport			:= 74,
	ActiveEnergyExport			:= 75,
	ReactiveEnergyTotal			:= 85,
	ReactiveEnergyInductive		:= 86,
	AReactiveEnergyCapacitive	:= 87,
	
	//Frequency
	FrequencyL1				:= 16,
	FrequencyL2				:= 17,
	FrequencyL3				:= 18,
	                           
	//Phase Angle              
	PhaseAngleL1			:= 19,
	PhaseAngleL2			:= 20,
	PhaseAngleL3			:= 21,
	
	//PowerFactor
	PowerFactorL1			:= 25,
	PowerFactorL2			:= 26,
	PowerFactorL3			:= 27
) USINT;
END_TYPE

// ---- POUs/Functions-FBs-Programs/IO_modules/Wago/Structs/Wago750495/eWago750495_HarmonicsDataID.TcDUT
{attribute 'qualified_only'}
{attribute 'strict'}
{attribute 'to_String'}
TYPE eWago750495_HarmonicsDataID :
(
	Current_RMS 		:= 001,
	Voltage_RMS 		:= 002,
	CurrentTHD			:= 003,
	VoltageTHD			:= 004
	
	//harmonics not declared for now
);
END_TYPE

// ---- POUs/Functions-FBs-Programs/IO_modules/Wago/Structs/Wago750495/eWago750495_MeasureGroupID.TcDUT
{attribute 'qualified_only'}
{attribute 'strict'}
{attribute 'to_String'}
TYPE eWago750495_MeasureGroupID :
(
	ac := 10,
	harmonicsL1 := 20,
	harmonicsL2 := 21,
	harmonicsL3	:= 22
) USINT;
END_TYPE

// ---- POUs/Functions-FBs-Programs/IO_modules/Wago/Structs/Wago750495/eWago750495_StatDataID.TcDUT
{attribute 'qualified_only'}
{attribute 'strict'}
TYPE eWago750495_StatDataID :
(
	Phase1 := 0,
	Phase2 := 1,
	Phase3 := 2,
	IOmodule:= 3
)USINT;
END_TYPE

// ---- POUs/Functions-FBs-Programs/IO_modules/Wago/Structs/Wago750495/ST_Wago750495_Data.TcDUT
TYPE ST_Wago750495_Data :
STRUCT
	//Voltages
	ar_VoltageLN					: ARRAY [0..3] OF REAL;
	ar_VoltageLL					: ARRAY [0..3] OF REAL;
	                            	      
	//Currents 
	ar_CurrentRMS					: ARRAY [0..4] OF REAL;                 	      
	                            	      
	//Power
	ar_ActivePower					: ARRAY [0..3] OF REAL;
	ar_ReactivePower				: ARRAY [0..3] OF REAL;
	ar_ApparentPower				: ARRAY [0..3] OF REAL;                     	      
	
	//Energy
	r_ActiveEnergyTotal				: REAL;
	r_ActiveEnergyImport			: REAL;
	r_ActiveEnergyExport			: REAL;
	r_ReactiveEnergyTotal			: REAL;
	r_ReactiveEnergyInductive		: REAL;
	r_AReactiveEnergyCapacitive		: REAL;
	
	//Frequency
	ar_Frequency					: ARRAY [0..3] OF REAL;
	                        		      
	//Phase Angle 
	ar_PhaseAngle					: ARRAY [0..3] OF REAL;          		      
	                        		      
	//PowerFactor     
	ar_Powerfactor					: ARRAY [0..3] OF REAL;      		      
	
	
END_STRUCT
END_TYPE

// ---- POUs/Functions-FBs-Programs/IO_modules/Wago/Structs/Wago750495/ST_Wago750495_ExtStatusWord.TcDUT
TYPE ST_Wago750495_ExtStatusWord :
STRUCT
	b_IncreasedMeasErr			: BOOL; //Stat 1 query L1,L2,L3:: increase measurement error of selected phase
	b_CurrentClipping			: BOOL; //Stat 2 query L1,L2,L3:: current out of measurable range of selected phase
	b_VoltageClipping			: BOOL; //Stat 3 query L1,L2,L3:: voltage out of measurable range of selected phase
	b_NoZeroCrossings			: BOOL; //Stat 4 query L1,L2,L3:: Zero Crossings missing of selected phase
	b_OverCurrent				: BOOL; //Stat 5 query L1,L2,L3:: Overcurrent of selected phase
	b_OverVoltage				: BOOL; //Stat 6- query L1,L2,L3: OverVoltage of selected phase.
	b_RotaryField				: BOOL; //Stat 6- query IO: 0:Clockwise, 1: counterclockwise
	b_UnderVoltage				: BOOL; //Stat 7- query L1,L2,L3: UnderVoltage of selected phase

END_STRUCT
END_TYPE

// ---- POUs/Functions-FBs-Programs/IO_modules/Wago/Structs/Wago750495/ST_Wago750495_Get.TcDUT
TYPE ST_Wago750495_Get :
STRUCT
	StatusWord				: ST_Wago750495_StatusWord;
	ExtStatusWord			: ST_Wago750495_ExtStatusWord;
	Data					: ST_Wago750495_Data;
END_STRUCT
END_TYPE

// ---- POUs/Functions-FBs-Programs/IO_modules/Wago/Structs/Wago750495/ST_Wago750495_Set.TcDUT
TYPE ST_Wago750495_Set :
STRUCT
	b_EnableRegisterComm		: BOOL;
	e_statusQuery				: eWago750495_StatDataID; //0: status L1, 1: status L2, 2: Status L3, 3: Status IO Module			
END_STRUCT
END_TYPE

// ---- POUs/Functions-FBs-Programs/IO_modules/Wago/Structs/Wago750495/ST_Wago750495_StatusWord.TcDUT
TYPE ST_Wago750495_StatusWord :
STRUCT
	b_ComFb						: BOOL; // 0: process Data, 1: Register Data
	b_Error						: BOOL; // 0: OK, 1: Error
	b_Error_IO					: BOOL; // 0: OK, 1: Error
	b_Error_L3					: BOOL; // 0: OK, 1: Error
	b_Error_L2					: BOOL; // 0: OK, 1: Error
	b_Error_L1					: BOOL; // 0: OK, 1: Error
	e_StatIDfb					: eWago750495_StatDataID;
	b_Warning					: BOOL; // 0: OK, 1: Transient reaction measured value collection active
	b_Cal						: BOOL; // 0: Measurement Mode, 1: Calibration Mode
	b_Over_1					: BOOL; // 0: OK, 1: Out Of Range
	b_Over_2					: BOOL; // 0: OK, 1: Out Of Range
	b_Over_3					: BOOL; // 0: OK, 1: Out Of Range
	b_Over_4					: BOOL; // 0: OK, 1: Out Of Range
	e_GroupID					: eWago750495_MeasureGroupID;

END_STRUCT
END_TYPE

// ---- POUs/MonitoringControl/HMI/_Structs/ControlStructures/OperationVars/ST_OperationVars.TcDUT
TYPE ST_OperationVars :
STRUCT
		inputgrid				: ST_OperationVars_Grid;
		Genset					: ST_OperationVars_Genset;
		PSB						: ST_OperationVars_Grid;
		charger					: ST_OperationVars_DCcharger;
		system					: ST_OperationVars_System;
		parallel				: ST_OperationVars_ParallelOperation;	
		BMS						: ST_OperationVars_BMS;	
END_STRUCT
END_TYPE

// ---- POUs/MonitoringControl/HMI/_Structs/ControlStructures/OperationVars/ST_OperationVars_BMS.TcDUT
TYPE ST_OperationVars_BMS :
STRUCT
	b_ManualStartHVDC	: BOOL;
END_STRUCT
END_TYPE

// ---- POUs/MonitoringControl/HMI/_Structs/ControlStructures/OperationVars/ST_OperationVars_DCcharger.TcDUT
TYPE ST_OperationVars_DCcharger :
STRUCT
	b_StartCharging						: BOOL;
	b_ResetCharger						: BOOL;
END_STRUCT
END_TYPE

// ---- POUs/MonitoringControl/HMI/_Structs/ControlStructures/OperationVars/ST_OperationVars_Genset.TcDUT
TYPE ST_OperationVars_Genset :
STRUCT 
	b_manualStart			: BOOL;
END_STRUCT
END_TYPE

// ---- POUs/MonitoringControl/HMI/_Structs/ControlStructures/OperationVars/ST_OperationVars_Grid.TcDUT
TYPE ST_OperationVars_Grid:
STRUCT
	b_SyncClose							: BOOL;
END_STRUCT
END_TYPE

// ---- POUs/MonitoringControl/HMI/_Structs/ControlStructures/OperationVars/ST_OperationVars_ParallelOperation.TcDUT
TYPE ST_OperationVars_ParallelOperation :
STRUCT
	b_DetectSlaves					: BOOL;
	
	
	// VDL ONLY
	r_ActivePowerSlave1				: REAL;
	r_ReactivePowerSlave1			: REAL;
	r_ActivePowerSlave2				: REAL;
	r_ReactivePowerSlave2			: REAL;
END_STRUCT
END_TYPE

// ---- POUs/MonitoringControl/HMI/_Structs/ControlStructures/OperationVars/ST_OperationVars_System.TcDUT
TYPE ST_OperationVars_System :
STRUCT
	//Powerstack
	r_NominalVoltage				: REAL := Settings.GridParams.r_GridNominalVoltage; //VAC
	r_NominalFrequency				: REAL := Settings.GridParams.r_GridNominalFrequency; //Hz
	
	//Power setpoints
	r_Pset							: REAL;// active power setpoint
	r_Qset							: REAL;// reactive power setpoint
	r_PFset							: REAL := 1;// powerfactor -1 .. 1
	b_PFsetEnable					: BOOL := TRUE;
	
	b_SounderMute					: BOOL;
	b_SounderTest					: BOOL;	
	
	//Mode transition
	b_GenGridModeTrans				: BOOL;	
	b_GridTakeOverEnable			: BOOL;
END_STRUCT
END_TYPE

// ---- POUs/MonitoringControl/HMI/_Structs/ControlStructures/ST_ControlsHMIonly.TcDUT
TYPE ST_ControlsHMIonly:
STRUCT
	b_Pup							: BOOL;
	b_Pdown							: BOOL;
	b_Qup							: BOOL;
	b_Qdown							: BOOL;
	b_QReset						: BOOL;
	b_PReset						: BOOL;
	b_HMITaskKill					: BOOL;
	b_ActivateSetting				: BOOL;
END_STRUCT
END_TYPE

// ---- POUs/MonitoringControl/HMI/_Structs/ControlStructures/ST_ControlVars.TcDUT
TYPE ST_ControlVars :
STRUCT
	b_start							: BOOL;
	b_stop							: BOOL;
	b_shutdown						: BOOL;
	b_Reset							: BOOL;
	b_SystemShutdown				: BOOL;
	b_EMstop						: BOOL;
	b_ClearHistory					: BOOL;
	b_ActivateSettings 				: BOOL;
	b_ActivateIotSettings			: BOOL;
	b_startDeHum					: BOOL;
END_STRUCT
END_TYPE

// ---- POUs/MonitoringControl/HMI/_Structs/MonitoringStructures/ST_HMIdata.TcDUT
TYPE ST_HMIdata :
STRUCT
	s_Type		: STRING(12);
	s_Name		: STRING(25);
	s_Data		: STRING(12);
	s_Unit		: STRING(4);
	b_Warning	: BOOL; 
END_STRUCT
END_TYPE

// ---- POUs/MonitoringControl/HMI/_Structs/MonitoringStructures/ST_HMI_ConditionalFormatting.TcDUT
TYPE ST_HMI_ConditionalFormatting :
STRUCT
	b_ShowPset			: BOOL;
	b_ShowQset			: BOOL;
	b_showPFset			: BOOL;
	b_ShowInputDisconnect: BOOL;
	b_ShowGenManStartStop: BOOL;
	b_ShowShowGensetInfo : BOOL;
	b_EnableTNCheckBox 		: BOOL;
	b_ShowExtgenset		: BOOL;
	b_TransportModeActive : BOOL;
	b_ShowGensetHybridMode: BOOL;
	b_showPSBData			: BOOL;
	b_showModetransbutton	: BOOL;
END_STRUCT
END_TYPE

// ---- POUs/MonitoringControl/HMI/_Structs/MonitoringStructures/ST_HMI_Monitor_AcDcCharger.TcDUT
TYPE ST_HMI_Monitor_AcDcCharger :
STRUCT
	state 			: STRING;
	available 		: BOOL;
	r_AcCurrentMax	: REAL;
	r_AcPowerMax	: REAL;
	r_DcPower 		: REAL;
	r_AcPower 		: REAL;
	r_AcCurrent		: REAL;
	r_AcVoltage		: REAL;
END_STRUCT
END_TYPE

// ---- POUs/MonitoringControl/HMI/_Structs/MonitoringStructures/ST_HMI_Monitor_Arraydata.TcDUT
TYPE ST_HMI_Monitor_Arraydata :
STRUCT
	ACInputData			: ARRAY [1..35] OF ST_HMIData;
	ACOutputData		: ARRAY [1..36] OF ST_HMIData;
	AcDcChargerData		: ARRAY [1..13] OF ST_HMIData;
	DcExtension			: ARRAY [1..4] OF ST_HMIData;
	PowerstackData 		: ARRAY [1..20] OF ST_HMIData;
	PmMasterData		: ARRAY [1..58] OF ST_HMIData;
	PmSlaveData			: ARRAY [1..58] OF ST_HMIData;
	PNcontrolData		: ARRAY [1..45] OF ST_HMIData;
	IotcontrolData		: ARRAY [1..45] OF ST_HMIData;
	PSBdata				: ARRAY [1..24] OF ST_HMIData;
	MBMUdata			: ARRAY [1..20] OF ST_HMIData;
	SBMU1Data			: ARRAY [1..21] OF ST_HMIData;
	SBMU2Data			: ARRAY [1..21] OF ST_HMIData;
	SBMU3Data			: ARRAY [1..21] OF ST_HMIData;
	SBMU4Data			: ARRAY [1..21] OF ST_HMIData;
	CoolingSystem		: ARRAY [1..5] OF ST_HMIData;
	CoolingSystemHp1	: ARRAY [1..10] OF ST_HMIData;
	CoolingSystemHp2	: ARRAY [1..10] OF ST_HMIData;
	Genset				: ARRAY [1..14] OF ST_HMIData;
END_STRUCT
END_TYPE

// ---- POUs/MonitoringControl/HMI/_Structs/MonitoringStructures/ST_HMI_Monitor_ArrayDataFormat.TcDUT
TYPE ST_HMI_Monitor_ArrayDataFormat :
STRUCT
	s_name				: STRING(25);
	s_type				: STRING(12);
	s_unit				: STRING(12);
	r_data				: REAL;
	i_precision			: INT := -1;
	b_warning			: BOOL;
END_STRUCT
END_TYPE

// ---- POUs/MonitoringControl/HMI/_Structs/MonitoringStructures/ST_HMI_Monitor_Connections.TcDUT
TYPE ST_HMI_Monitor_Connections :
STRUCT
	b_ExtControllerEnabled		: BOOL;
	e_ExtConnectionState		: eConnectionState;
	s_OutputJson				: STRING(2000);
	b_IoTEnabled				: BOOL;
	e_IoTConnectionState		: eConnectionState;
	b_PsbOK						: BOOL;			
	e_ActiveController			: eControlSources;
	e_ProfinetState				: eNetcomState;
	e_EthercatState				: eNetcomState;
	r_CPUload					: REAL;
	
END_STRUCT
END_TYPE

// ---- POUs/MonitoringControl/HMI/_Structs/MonitoringStructures/ST_HMI_Monitor_Battery.TcDUT
TYPE ST_HMI_Monitor_Battery :
STRUCT
	e_status			: eBMS_Status;
	r_SocScaled			: REAL := 10; 
	r_SoCReal			: REAL;
	r_CellVoltageMax	: REAL;
	r_CellVoltageMin	: REAL;
	r_CellTempMax		: REAL;
	r_CellTempMin		: REAL;
	r_MaxDischargePower	: REAL;
	r_MaxChargePower	: REAL;
	r_DCvoltage			: REAL;
	r_DCcurrent			: REAL;
	r_SoH				: REAL;
	r_NetRemainingCapacity: REAL; //kWh
	ui_CycleCount		: UINT;
	
END_STRUCT
END_TYPE

// ---- POUs/MonitoringControl/HMI/_Structs/MonitoringStructures/ST_HMI_Monitor_CoolingSystem.TcDUT
TYPE ST_HMI_Monitor_CoolingSystem :
STRUCT
	e_OperationMode 		: eCoolingSystemState;
	e_HeatPumpStatus		: eHeatPumpState;
	r_CoolantTemperature	:	REAL;
	r_CoolantPressure		:	REAL;
	r_EnclosureDewpoint		:	REAL;
	b_HeatPumpError			: 	BOOL;
	b_HeatPumpWarning		:	BOOL;
	b_CoolantPressureWarning: 	BOOL;
	b_CoolantPressureError	:	BOOL;
	b_CoolantTempWarning	: 	BOOL;
END_STRUCT
END_TYPE

// ---- POUs/MonitoringControl/HMI/_Structs/MonitoringStructures/ST_HMI_Monitor_Enclosure.TcDUT
TYPE ST_HMI_Monitor_Enclosure :
STRUCT
	//Doors
	b_DoorClosedClientPanel		: BOOL;
	b_DoorClosedControlPanel	: BOOL;
	b_DoorClosedInverter		: BOOL;
	
	//climate
	r_Humidity					: REAL := -255;
	r_Temperature				: REAL := -255;
	b_HumidityHigh				: BOOL;
	b_HumidityTooHigh			: BOOL;
	b_TemperatureHigh			: BOOL;
	b_TemperatureTooHigh		: BOOL;
	b_TemperatureLow			: BOOL;
	b_TemperatureTooLow			: BOOL;
	
END_STRUCT
END_TYPE

// ---- POUs/MonitoringControl/HMI/_Structs/MonitoringStructures/ST_HMI_Monitor_FireDetection.TcDUT
TYPE ST_HMI_Monitor_FireDetection :
STRUCT
	e_SmokeDetectorState			: eSmokeDetectAlarmStatus;
	e_CoDetectorState				: eCOAlarmStatus;
	r_CoDetectorLeftValue			: REAL; //ppm
	r_CoDetectorRightValue			: REAL; //ppm			
END_STRUCT
END_TYPE

// ---- POUs/MonitoringControl/HMI/_Structs/MonitoringStructures/ST_HMI_Monitor_IPSU.TcDUT
TYPE ST_HMI_Monitor_IPSU :
STRUCT
	b_24VdcOK			: BOOL;
	b_400VacOK			: BOOL;
	b_HvdcOK			: BOOL;
	b_GridFuseOK		: BOOL;
	b_CeeFuseOK			: BOOL;
	e_400VSource		: e400VSupplySource;
END_STRUCT
END_TYPE

// ---- POUs/MonitoringControl/HMI/_Structs/MonitoringStructures/ST_HMI_Monitor_Limits.TcDUT
TYPE ST_HMI_Monitor_Limits :
STRUCT
	//LIMITS
	//r_Pmin						: REAL ;
	//r_Pmax						: REAL ;
	//r_QMin						: REAL ;
	//r_QMax						: REAL ;
	r_ACcurrentLimit			: REAL;
	r_ApparentPowerlimit		: REAL;
	r_ActivePowerlimit			: REAL;
	r_DCcurrentLimit			: REAL;
	r_DroopLimit				: REAL;
	
END_STRUCT
END_TYPE

// ---- POUs/MonitoringControl/HMI/_Structs/MonitoringStructures/ST_HMI_Monitor_OCP.TcDUT
TYPE ST_HMI_Monitor_OCP : //overcurrent protection
STRUCT
	b_InputMCCBstate			: BOOL;
	b_OutputMCCBstate			: BOOL;
	b_InputOverloadWarning		: BOOL;
	b_InputOverloadAlarm		: BOOL;
	b_OutputOverloadWarning		: BOOL;
	b_OutputOverloadAlarm		: BOOL;
	s_Location					: STRING;
	r_CurrentPeak				: REAL;
	t_PeakDuration				: TIME;	
END_STRUCT
END_TYPE

// ---- POUs/MonitoringControl/HMI/_Structs/MonitoringStructures/ST_HMI_Monitor_Powerstack.TcDUT
TYPE ST_HMI_Monitor_Powerstack :
STRUCT
	// stack
	r_Powerload					: REAL;
	r_DcPower					: REAL;
	r_ActivePower				: REAL;
	r_throttlingValue			: REAL;
	
	b_ACDetected				: BOOL;
	b_DCDetected				: BOOL;
	b_StartedState				: BOOL;
	b_islandOperation			: BOOL;
	b_ControlEnabled			: BOOL;
	e_NetContState				: eNetContactorState;
	e_ACrotationState			: eACRotationState;
	e_StatusPowerStack			: eStatusPowerstack;
	
	//Master
	b_MasterEnabled				: BOOL;
	b_MasterWarning				: BOOL;
	b_MasterMCCBfb				: BOOL;
	e_MasterState				: eStatusPowerModule;
	r_MasterthrotValue			: REAL;
	b_MasterTempThrotActive		: BOOL;
	b_MasterCurrThrotActive		: BOOL;		
	
	
	b_SlaveEnabled				: BOOL;
	b_SlaveWarning				: BOOL;
	b_SlaveMCCBfb				: BOOL;
	e_SlaveState				: eStatusPowerModule;
	r_SlavethrotValue			: REAL;
	b_SlaveTempThrotActive		: BOOL;
	b_SlaveCurrThrotActive		: BOOL;		
	
END_STRUCT
END_TYPE

// ---- POUs/MonitoringControl/HMI/_Structs/MonitoringStructures/ST_HMI_Monitor_Protections.TcDUT
TYPE ST_HMI_Monitor_Protections :
STRUCT
	b_MrcdbOK					: BOOL;
	b_MrcdbWarning				: BOOL;
	b_MrcdbAlarm				: BOOL;
	b_InsulationEnable			: BOOL;
	b_InsulationOk				: BOOL;
	b_InsulationWarning			: BOOL;
	b_InsulationAlarm			: BOOL;
	b_InsulationPenDetected		: BOOL; //discrepence of PEN config and detected situation
	e_EarthingSystemDetected	: eEarthingSystems; //0: Unknown, 1: TN-S, 2: TN-C, 3: IT.
	b_SurgeType12OK				: BOOL;
	b_SurgeType3OK				: BOOL;
END_STRUCT
END_TYPE

// ---- POUs/MonitoringControl/HMI/_Structs/MonitoringStructures/ST_HMI_Monitor_PSB.TcDUT
TYPE ST_HMI_Monitor_PSB :
STRUCT
	b_Connected : BOOL;
	b_Active	: BOOL;
END_STRUCT
END_TYPE

// ---- POUs/MonitoringControl/HMI/_Structs/MonitoringStructures/ST_HMI_Monitor_switchgear.TcDUT
TYPE ST_HMI_Monitor_switchgear :
STRUCT
	//Switchgear
	b_ACDetectedBusbar			: BOOL;
	b_ACDetectedInput			: BOOL;
	b_DCDetected				: BOOL;
	b_PeNeutralLink				: BOOL;
	b_ACInputState				: BOOL; //summary of MCCB and contactor state.
	b_InputSync					: BOOL;
	r_ACInputPower				: REAL;
	b_NetContactorState			: BOOL; //summary of netcontactor left and right close state.
	b_ACOutputState				: BOOL;
	r_ACOutputPower				: REAL; 
	b_DCCouplingState			: BOOL;
	r_DCCouplingCurrent			: REAL;
END_STRUCT
END_TYPE

// ---- POUs/MonitoringControl/HMI/_Structs/MonitoringStructures/ST_HMI_Monitor_System.TcDUT
TYPE ST_HMI_Monitor_System :
STRUCT
	r_currentEfficiency		: REAL;
	r_averageEfficiency		: REAL;
	r_RountripEfficiency	: REAL;
	r_DischargeEnergy		: REAL;
	r_ChargedEnergy			: REAL;
	
	e_SystemState			: eSystemState; //0:Idle, 1: Stand-by, 2:Conditioning, 3:Dry-Cycle, 4: Running, 5: Charging only, 6: Discharging only, 7: Stopped 8:Fault
	e_GridMode				: eGridmode;
	e_UgridPowermode		: eUgridPowermode;
	
	b_EarthingSelected		: BOOL;
	b_startAllowed			: BOOL;
	
	b_Alert					: BOOL;
	b_SMSnumberConfigured	: BOOL;
	b_CustomNameConfigured	: BOOL;
	b_TransportModePending	: BOOL;
	b_MasterSlaveModeEnabled: BOOL;
	
	s_SystemName			: STRING(20);
END_STRUCT
END_TYPE

// ---- POUs/MonitoringControl/HMI/_Structs/MonitoringStructures/ST_HMI_Monitor_UPS.TcDUT
TYPE ST_HMI_Monitor_UPS :
STRUCT
	b_ChargerActive		: BOOL;
	b_SupplyOnBattery	: BOOL;
	r_InputVoltage		: REAL;
	r_OutputVoltage		: REAL;
	r_OutputCurrent		: REAL;
	r_BatteryVoltage	: REAL;
	b_InputVoltageFault	: BOOL;
	b_BatteryLowInfo	: BOOL;
	b_BatteryLowWarning : BOOL;
	b_BatteryLowCritical: BOOL;
	ui_SoC				: UINT;
END_STRUCT
END_TYPE

// ---- POUs/MonitoringControl/HMI/_Structs/MonitoringStructures/ST_HMI_Monitor_ZPT.TcDUT
TYPE ST_HMI_Monitor_ZPT :
STRUCT
	b_ZPTOverloadWarning	: BOOL;
	b_ZPTOverloadAlarm		: BOOL;
	b_VoltageUnbalanceWarning: BOOL;
	b_VoltageUnbalanceAlarm	: BOOL;
	r_TemperatureL1			: REAL;
	b_TempWarningL1			: BOOL;
	b_TempAlarmL1			: BOOL;
	r_TemperatureL2			: REAL;
	b_TempWarningL2			: BOOL;
	b_TempAlarmL2			: BOOL;
	r_TemperatureL3			: REAL;
	b_TempWarningL3			: BOOL;
	b_TempAlarmL3			: BOOL;
	r_powerload				: REAL;	//%
	r_voltageunbalance		: REAL; //%
END_STRUCT
END_TYPE

// ---- POUs/MonitoringControl/HMI/_Structs/MonitoringStructures/ST_HMI_PowerMeas.TcDUT
TYPE ST_HMI_PowerMeas :
STRUCT
	Voltage			: REAL;
	Frequency		: REAL;
	ActivePower		: REAL;
	ReactivePower	: REAL;
	Current			: REAL;
END_STRUCT
END_TYPE

// ---- POUs/MonitoringControl/HMI/_Structs/MonitoringStructures/ST_HMI_PowerMeasDC.TcDUT
TYPE ST_HMI_PowerMeasDC :
STRUCT
	Voltage : REAL;
	Current	: REAL;
	Power	: REAL;
	SOC		: REAL;
END_STRUCT
END_TYPE

// ---- POUs/MonitoringControl/HMI/_Structs/ST_HMI_Control.TcDUT
TYPE ST_HMI_Control EXTENDS ST_System_Control:
STRUCT
	HMIonly				: ST_ControlsHMIonly;
END_STRUCT
END_TYPE

// ---- POUs/MonitoringControl/HMI/_Structs/ST_HMI_Historize.TcDUT
TYPE ST_HMI_Historize :
STRUCT
	PSB				: ST_HMI_PowerMeas;
	Input			: ST_HMI_PowerMeas;
	Output			: ST_HMI_PowerMeas;
	Inverter		: ST_HMI_PowerMeas;
	Battery			: ST_HMI_PowerMeasDC;
	Charger			: ST_HMI_PowerMeas;
	DcCoupling		: ST_HMI_PowerMeasDC;
END_STRUCT
END_TYPE

// ---- POUs/MonitoringControl/HMI/_Structs/ST_HMI_Monitor.TcDUT
//CHANGING THESE VARIABLES WILL RESULT IN BROKEN LINKS TO THE HMI!
TYPE ST_HMI_Monitor :
STRUCT
	ConditionalFormatting		: ST_HMI_ConditionalFormatting;
	System						: ST_HMI_Monitor_System;
	Powerstack					: ST_HMI_Monitor_Powerstack;
	enclosure					: ST_HMI_Monitor_enclosure;
	firedetection				: ST_HMI_Monitor_Firedetection;
	IPSU						: ST_HMI_Monitor_IPSU;
	OCP							: ST_HMI_Monitor_OCP;
	UPS							: ST_HMI_Monitor_UPS;
	protections					: ST_HMI_Monitor_protections;
	ZPT							: ST_HMI_Monitor_ZPT;
	Switchgear					: ST_HMI_Monitor_switchgear;
	Battery						: ST_HMI_Monitor_Battery;					
	Limits						: ST_HMI_Monitor_limits;
	Connections					: ST_HMI_Monitor_Connections;
	arraydata					: ST_HMI_Monitor_Arraydata;
	cooling						: ST_HMI_Monitor_CoolingSystem;
	AcDcCharger					: ST_HMI_Monitor_AcDcCharger;
	Powercontroller				: ST_PowerControl_Get;
	GenGridController			: ST_GenGridController_get;
	controlfb					: ST_ControlVars;
	PSB							: ST_HMI_Monitor_PSB;	
	b_testBool					: BOOL;
END_STRUCT
END_TYPE

// ---- POUs/MonitoringControl/IoT/DUTS/eConnectionState.TcDUT
{attribute 'qualified_only'}
{attribute 'strict'}
{attribute 'to_string'}
 
TYPE eConnectionState :
(
	disconnected := 0,			// no mqtt connection established
	connected	:= 1,			 // connected but not authorized yet
	authorization_declined := 2, // connected but authorization failed
	authorized	:= 3			// connected and authorized
);
END_TYPE

// ---- POUs/MonitoringControl/IoT/DUTS/eDataMappingVarNames.TcDUT
{attribute 'qualified_only'}
{attribute 'to_string'}

TYPE eDataMappingVarNames :
(*
 * Enumeration for mapping every variable in ST_System_Monitor to a fixed
 * monitoring ID.  The hierarchy is fully expanded at every nesting level.
 *
 * Naming convention:
 *   Structs : <topLevel>_<field>_<subField>_..._<leafField>
 *   Arrays  : <path>_<indexName>  where the index names are:
 *               _AVG      (index 0)
 *               _L1       (index 1)
 *               _L2       (index 2)
 *               _L3       (index 3)
 *               _N        (index 4)
 *               _minimum  (index 5)
 *               _maximum  (index 6)
 *   Only electrical measurement arrays are individually expanded:
 *   ar_ActivePower, ar_ReactivePower, ar_ApparentPower,
 *   ar_PhaseVoltage, ar_LineVoltage, ar_Current,
 *   ar_Frequency, ar_THD, ar_PowerFactor.
 *   The aggregate array variable is NOT included; only individual
 *   per-index entries are present (e.g. ar_Current_AVG, ar_Current_L1).
 *
 *)
(	
None													:= 0,
	(*═════════════════════════════════════════════════════════*)
	(*  Safety and System State    *)
	(*═════════════════════════════════════════════════════════*)
	safety_b_SafetyOK                                          , (* BOOL *)
	safety_b_EstopChannelAOK                                   , (* BOOL *)
	safety_b_EstopChannelBOK                                   , (* BOOL *)
	safety_b_InsulationMonitorOK                               , (* BOOL *)
	safety_b_MRCDBOK                                           , (* BOOL *)
	safety_b_InverterDoorOK                                    , (* BOOL *)
	safety_b_ZptOK                                             , (* BOOL *)
	system_b_SMSnumberConfigured                               , (* BOOL *)
	system_b_CustomNameConfigured                              , (* BOOL *)
	system_s_SystemName                                        , (* STRING(20) *)
	system_b_TransportModePending                              , (* BOOL *)
	system_b_DehumModePending                                  , (* BOOL *)
	system_e_State                                             , (* eSystemState *)
	system_e_gridmode                                          , (* eGridmode *)
	system_e_UgridPowermode                                    , (* eUgridPowermode *)
	system_b_StartAllowed                                      , (* BOOL *)
	system_r_CurrentEfficiency                                 , (* REAL *)
	system_r_AvgEfficiency                                     , (* REAL *)
	system_r_RoundtripEfficiency                               , (* REAL *)
	system_DT_SystemTime                                       , (* DT *)
	system_PowerController_r_CurrentAct                        , (* REAL *)
	system_PowerController_r_Sact                              , (* REAL *)
	system_PowerController_r_PAct                              , (* REAL *)
	system_PowerController_r_QAct                              , (* REAL *)
	system_PowerController_r_PhaseVoltageAct                   , (* REAL *)
	system_PowerController_r_PFact                             , (* REAL *)
	system_PowerController_r_FeedInCurrentLimitActual          , (* REAL *)
	system_PowerController_r_SupplyInCurrentLimitActual        , (* REAL *)
	system_PowerController_b_ThrottlingActive                  , (* BOOL *)
	system_PowerController_ui_ThrottlingType                   , (* UINT *)
	system_PowerController_events_b_ReactivePIDError           , (* BOOL *)
	system_PowerController_events_b_ActivePIDError             , (* BOOL *)
	system_PowerController_events_b_FreqShiftPIDError          , (* BOOL *)
	system_GenGridController_b_active                          , (* BOOL *)
	system_GenGridController_b_faultActive                     , (* BOOL *)
	system_GenGridController_b_gensetHot                       , (* BOOL *)
	system_GenGridController_b_gensetStarting                  , (* BOOL *)
	system_GenGridController_b_ModeTransActive                 , (* BOOL *)
	system_GenGridController_b_ModeTransInhibit                , (* BOOL *)
	system_GenGridController_b_ModeChanged                     , (* BOOL *)
	system_GenGridController_b_ShowModeTrans                   , (* BOOL *)
	system_GenGridController_b_extGensetMode                   , (* BOOL *)
	system_GenGridController_b_gensetcontrol                   , (* BOOL *)
	system_GenGridController_e_BreakerMode                     , (* eBreakerOperationMode *)
	system_GenGridController_e_PowerControlMode                , (* ePowerControlMode *)
	system_GenGridController_e_GensetMode                      , (* eGensetMode *)
	system_GenGridController_e_GensetStartStop                 , (* eGensetStartStop *)
	system_GenGridController_e_state                           , (* eGenGridState *)
	system_GenGridController_e_RunCondition                    , (* eRunCondition *)
	system_GenGridController_events_b_InvalidGensetParameters  , (* BOOL *)
	system_GenGridController_events_b_RotationFieldFault       , (* BOOL *)
	system_GenGridController_events_b_CurrentLimitDisconnect   , (* BOOL *)
	system_GenGridController_events_b_CurrentLimitTrip         , (* BOOL *)
	system_GenGridController_events_b_EmstopDisconnect         , (* BOOL *)
	system_GenGridController_events_b_ShutdownDisconnect       , (* BOOL *)
	system_GenGridController_events_b_OverloadTrip             , (* BOOL *)
	system_GenGridController_events_b_OverFreqTrip             , (* BOOL *)
	system_GenGridController_events_b_UnderFreqTrip            , (* BOOL *)
	system_GenGridController_events_b_OverVoltTrip             , (* BOOL *)
	system_GenGridController_events_b_UnderVoltTrip            , (* BOOL *)
	system_GenGridController_events_b_ShutdownTimeOut          , (* BOOL *)
	system_GenGridController_events_b_SynchronisationFault     , (* BOOL *)
	system_GenGridController_events_b_StartupFault             , (* BOOL *)
	system_GenGridController_events_b_WarmupFault              , (* BOOL *)
	system_GenGridController_events_b_GenDownTrip              , (* BOOL *)
	system_GenGridController_events_b_GridLostTrip             , (* BOOL *)
	system_GenGridController_events_b_TransToGenIsoInhibit     , (* BOOL *)
	system_GenGridController_events_b_TransToGenDroopInhibit   , (* BOOL *)
	system_GenGridController_events_b_TransToGenFixInhibit     , (* BOOL *)
	system_GenGridController_events_b_TransFromInputGridAckRQ  , (* BOOL *)
	system_GenGridController_events_b_TransFromInputGenAckRQ   , (* BOOL *)
	system_GenGridController_events_b_StartingInhibit          , (* BOOL *)
	system_events_b_RestartRequiredMachineName                 , (* BOOL *)
	system_events_b_TimeUpdateFailed                           , (* BOOL *)

